Staubli VAL3: loadmaster4.pgx

program loadmaster4(string x_sMasterFile4 (dimensions=1))
begin
  if master:libLoad(x_sMasterFile4)<0
    popUpMsg("nO ok")
  endIf
  frmaster[4].trsf=master:tTool.trsf
  //取个数
  nsize[4]=size(master:ptRoutingPath)
  //存个数
  resize(pdemo4,1,nsize[4])
  //保存程序
  master:libSave()
end
